{attribute 'TcCallAfterOutputUpdate'}
PROGRAM MAIN
VAR
	fbGetCurTaskIdx 			: GETCURTASKINDEX;
	bFirstCycle					: BOOL;
END_VAR

// =========================================================
	// Get plc task first cycle flag	
fbGetCurTaskIdx(); 
bFirstCycle:= _TaskInfo[fbGetCurTaskIdx.index].FirstCycle;

IF bFirstCycle THEN
	;
END_IF

// =========================================================

END_PROGRAM

(* stored: Version 1.1.0.1
   POU MAIN: Id {53e098ee-c10b-4533-88f1-a760e550a780}, SpecialFunc None *)
